Fanuc KAREL source: kd00057.KL

PROGRAM KD00057
%STACKSIZE=65535
%PRIORITY=65535
%NOLOCKGROUP
VAR
I : INTEGER
J : INTEGER
B : BOOLEAN
R : REAL
S : STRING[80]
P : POSITION
Q : POSITION
BEGIN
-- UNRESOLVED_PC line 13 opcodes [01 22 1C 06 22 1C 07 82 0B] marker_code=0
END KD00057
